TYPE ST_CURING_STATION_HMI :
STRUCT
	state:			ST_CURING_STATION_STATE;
	service:		ST_CURING_STATION_SERVICE;
	settings:		ST_CURING_STATION_SETTINGS;
	
	cyls:			ARRAY[0..1] OF ST_CYL_HMI;
	heater:			ST_CURING_STATION_HEATER_CONTROL_HMI;
	
	
END_STRUCT
END_TYPE

(* stored: Version 1.1.0.1
   DUT ST_CURING_STATION_HMI: Id {23ea0c5a-6f3c-4e26-9e32-58d17e3f60fa} *)
